// TIA Portal V20 export
TYPE "LER_typeAlignSyncMoveInterface"
// stored: Access Published
   STRUCT
      commands : "LER_typeAlignSyncMoveCommands";
      monitoring : "LER_typeAlignSyncMoveMonitoring";
      configuration : "LER_typeAlignSyncMoveConfiguration";
   END_STRUCT;
END_TYPE
